// TIA Portal V20 export
VAR_GLOBAL   // PLC tag table "PROFIDrive"
   LT3_OUT AT %Q11200.0 : "S_STW1";
   SL_IN AT %I11050.0 : "S_ZSW1";
   LT1_OUT AT %Q11100.0 : "S_STW1";
   CT2_OUT AT %Q10250.0 : "S_STW1";
   SL_OUT AT %Q11050.0 : "S_STW1";
   CT2_IN AT %I10250.0 : "S_ZSW1";
   LT4_IN AT %I11250.0 : "S_ZSW1";
   LT1_IN AT %I11100.0 : "S_ZSW1";
   CT1_OUT AT %Q10200.0 : "S_STW1";
   MH2_OUT AT %Q10150.0 : "S_STW1";
   MH1_OUT AT %Q10100.0 : "S_STW1";
   MH1_IN AT %I10100.0 : "S_ZSW1";
   LT2_IN AT %I11150.0 : "S_ZSW1";
   LT4_OUT AT %Q11250.0 : "S_STW1";
   LT2_OUT AT %Q11150.0 : "S_STW1";
   MH2_IN AT %I10150.0 : "S_STW1";
   LT3_IN AT %I11200.0 : "S_ZSW1";
   CT1_IN AT %I10200.0 : "S_ZSW1";
END_VAR
